// Mitsubishi GX Developer project: gate   PLC: FX1N

PROGRAM MAIN
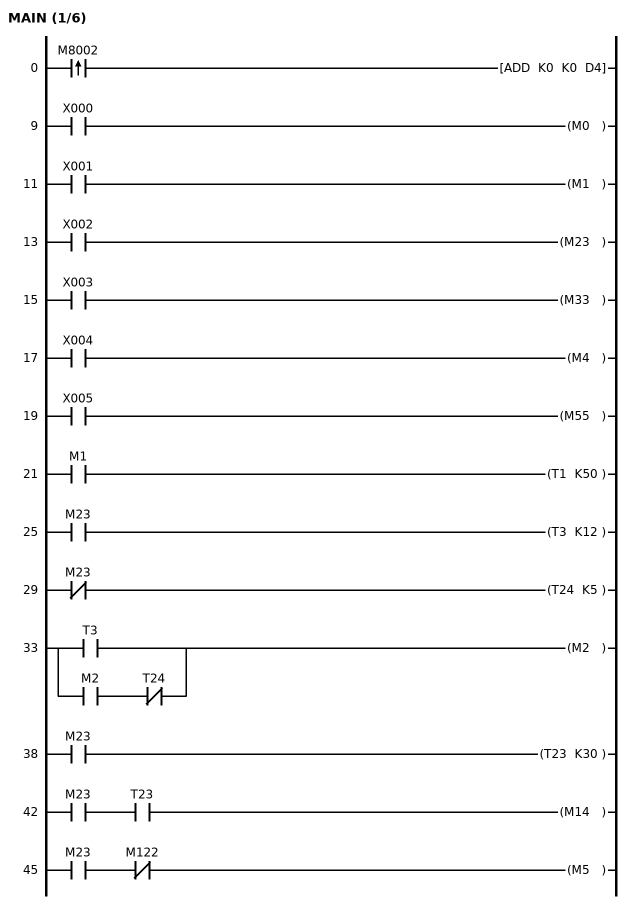
0     LDP     M8002
      ADD     K0 K0 D4
        [note] set car sensor to zero
9     LD      X000
      OUT     M0
        [note] external sw
11    LD      X001
      OUT     M1
        [note] internal sw
13    LD      X002
      OUT     M23
        [note] gate safety sw
15    LD      X003
      OUT     M33
        [note] car sensor
17    LD      X004
      OUT     M4
        [note] light on sensor
19    LD      X005
      OUT     M55
        [note] scrubber sensor
21    LD      M1
      OUT     T1 K50
        [note] internal open block delay
25    LD      M23
      OUT     T3 K12
        [note] X002 gate sensor
29    LDI     M23
      OUT     T24 K5
        [note] gate sensor debounse off
33    LD      T3
      LD      M2
      ANI     T24
      ORB
      OUT     M2
        [note] gate sensor debounce on
38    LD      M23
      OUT     T23 K30
        [note] car near gate timer
42    LD      M23
      AND     T23
      OUT     M14
        [note] car near gate
45    LD      M23
      ANI     M122
      OUT     M5
        [note] gate sensor and block
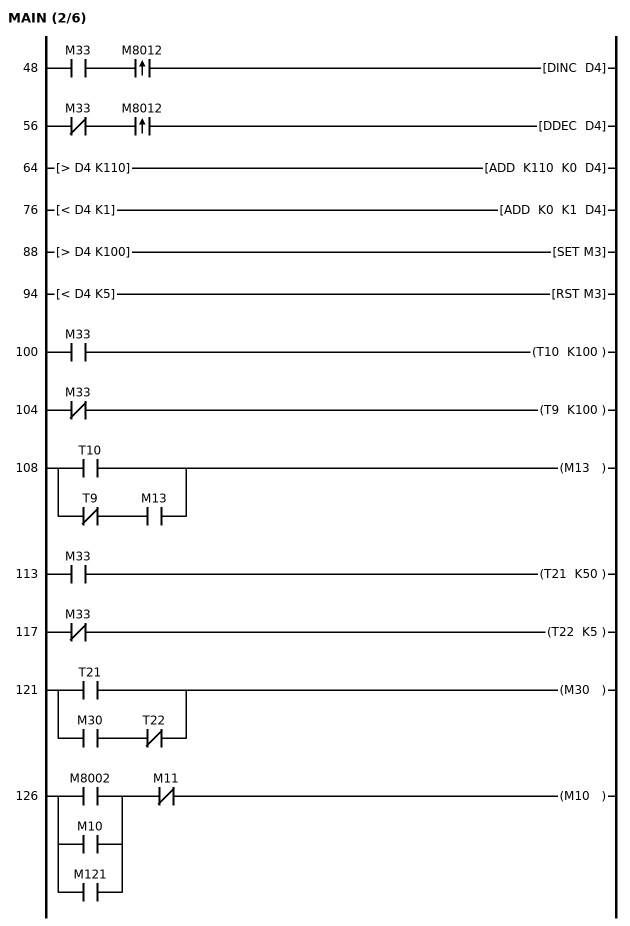
48    LD      M33
      ANDP    M8012
      DINC    D4
56    LDI     M33
      ANDP    M8012
      DDEC    D4
64    LD>     D4 K110
      ADD     K110 K0 D4
        [note] max limit  debounce car sensor
76    LD<     D4 K1
      ADD     K0 K1 D4
        [note] min limit  debounce car sensor
88    LD>     D4 K100
      SET     M3
94    LD<     D4 K5
      RST     M3
100   LD      M33
      OUT     T10 K100
        [note] x003  car sensor
104   LDI     M33
      OUT     T9 K100
        [note] debounce off
108   LD      T10
      LDI     T9
      AND     M13
      ORB
      OUT     M13
        [note] car sensor slow debounce
113   LD      M33
      OUT     T21 K50
        [note] car sensor fast  ON
117   LDI     M33
      OUT     T22 K5
        [note] car sensor fast OFF
121   LD      T21
      LD      M30
      ANI     T22
      ORB
      OUT     M30
        [note] car sensor fast
126   LD      M8002
      OR      M10
      OR      M121
      ANI     M11
      OUT     M10
        [note] ******** whaiting
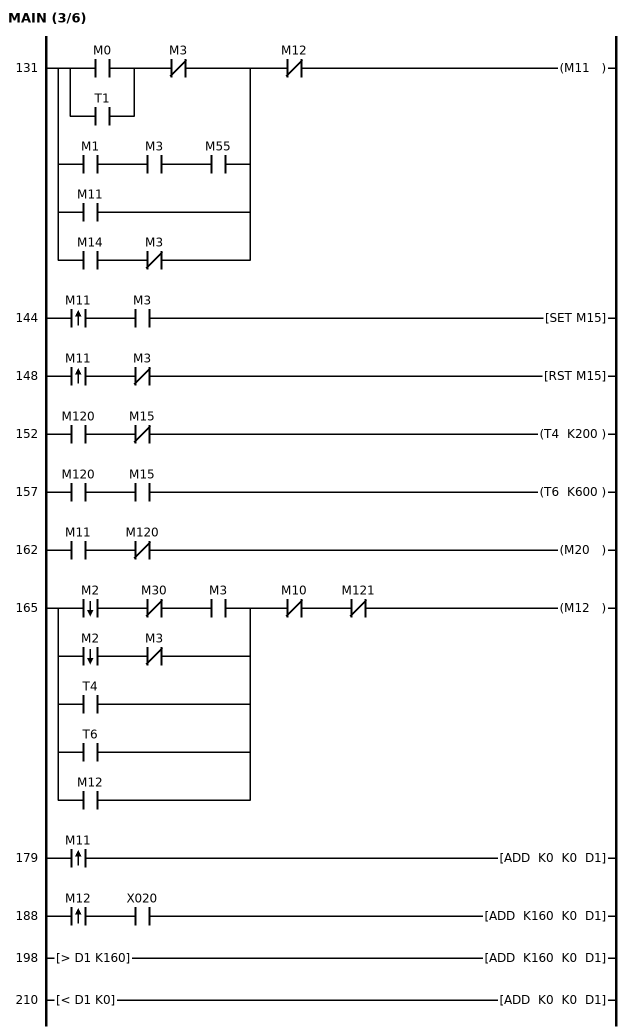
131   LD      M0
      OR      T1
      ANI     M3
      LD      M1
      AND     M3
      AND     M55
      ORB
      OR      M11
      LD      M14
      ANI     M3
      ORB
      ANI     M12
      OUT     M11
        [note] ******* entrance open begin
144   LDP     M11
      AND     M3
      SET     M15
        [note] car inside box
148   LDP     M11
      ANI     M3
      RST     M15
        [note] car outside box
152   LD      M120
      ANI     M15
      OUT     T4 K200
        [note] waiting entranñe
157   LD      M120
      AND     M15
      OUT     T6 K600
        [note] exit waiting
162   LD      M11
      ANI     M120
      OUT     M20
165   LDF     M2
      ANI     M30
      AND     M3
      LDF     M2
      ANI     M3
      ORB
      OR      T4
      OR      T6
      OR      M12
      ANI     M10
      ANI     M121
      OUT     M12
        [note] ******* entrance close begin
179   LDP     M11
      ADD     K0 K0 D1
        [note] set gate open start pos
188   LDP     M12
      AND     X020
      ADD     K160 K0 D1
        [note] set gate close start pos
198   LD>     D1 K160
      ADD     K160 K0 D1
        [note] gate up limit
210   LD<     D1 K0
      ADD     K0 K0 D1
        [note] gate close limit
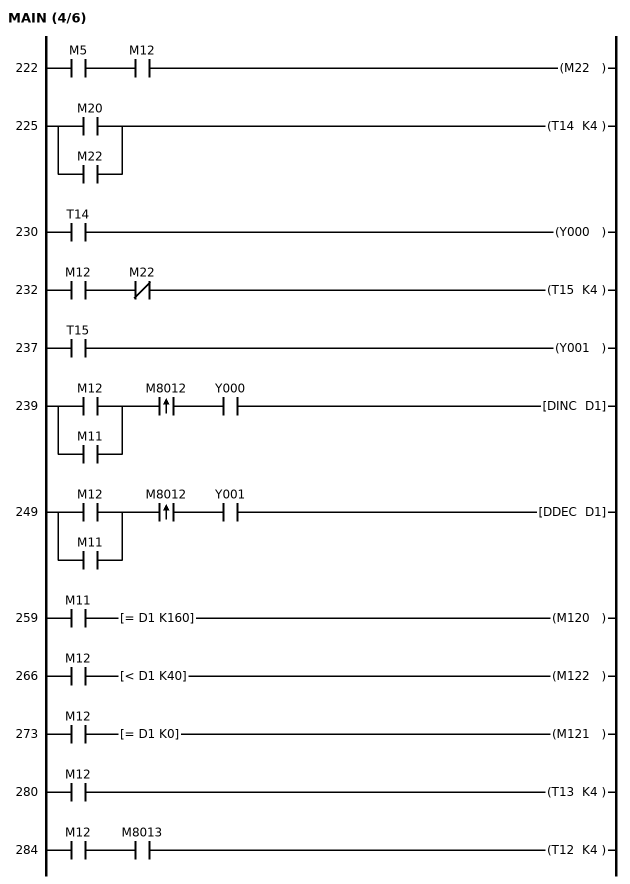
222   LD      M5
      AND     M12
      OUT     M22
        [note] open in close
225   LD      M20
      OR      M22
      OUT     T14 K4
        [note] gears safety time
230   LD      T14
      OUT     Y000
        [note] out relay block * open signal
232   LD      M12
      ANI     M22
      OUT     T15 K4
        [note] gears safety timer
237   LD      T15
      OUT     Y001
        [note] gate close output
239   LD      M12
      OR      M11
      ANDP    M8012
      AND     Y000
      DINC    D1
        [note] gate open timer incr
249   LD      M12
      OR      M11
      ANDP    M8012
      AND     Y001
      DDEC    D1
        [note] gate close timer decr
259   LD      M11
      AND=    D1 K160
      OUT     M120
        [note] open end
266   LD      M12
      AND<    D1 K40
      OUT     M122
        [note] block M5 and pic-pic
273   LD      M12
      AND=    D1 K0
      OUT     M121
        [note] close end
280   LD      M12
      OUT     T13 K4
        [note] close  pik
284   LD      M12
      AND     M8013
      OUT     T12 K4
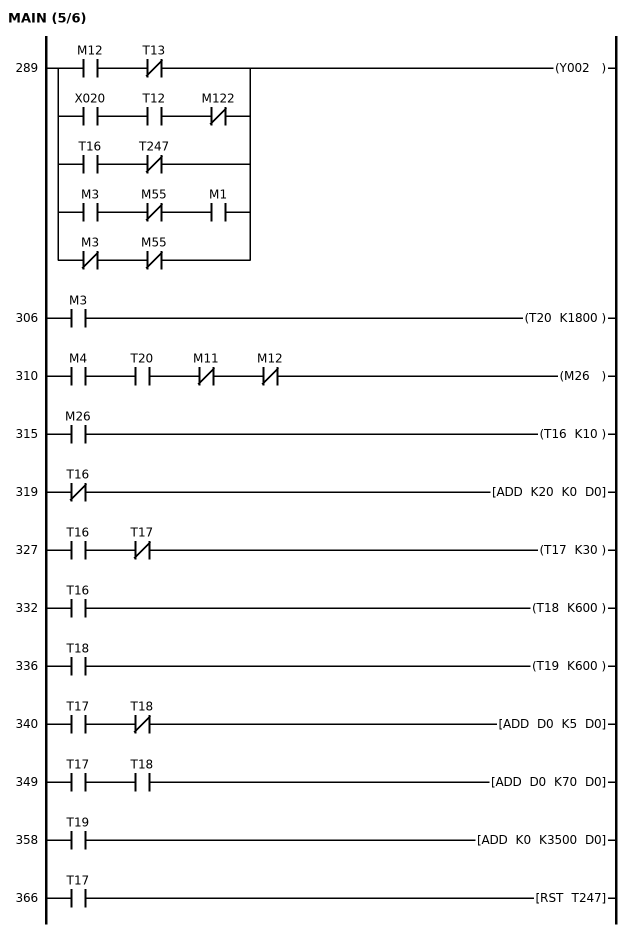
289   LD      M12
      ANI     T13
      LD      X020
      AND     T12
      ANI     M122
      ORB
      LD      T16
      ANI     T247
      ORB
      LD      M3
      ANI     M55
      AND     M1
      ORB
      LDI     M3
      ANI     M55
      ORB
      OUT     Y002
        [note] siren
306   LD      M3
      OUT     T20 K1800
        [note] block get-out entrance
310   LD      M4
      AND     T20
      ANI     M11
      ANI     M12
      OUT     M26
        [note] *** warning begin ****
315   LD      M26
      OUT     T16 K10
319   LDI     T16
      ADD     K20 K0 D0
327   LD      T16
      ANI     T17
      OUT     T17 K30
332   LD      T16
      OUT     T18 K600
        [note] 1 min timer
336   LD      T18
      OUT     T19 K600
340   LD      T17
      ANI     T18
      ADD     D0 K5 D0
349   LD      T17
      AND     T18
      ADD     D0 K70 D0
358   LD      T19
      ADD     K0 K3500 D0
366   LD      T17
      RST     T247
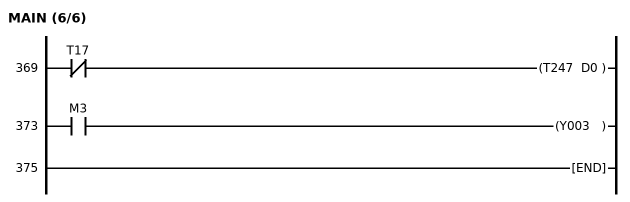
369   LDI     T17
      OUT     T247 D0
373   LD      M3
      OUT     Y003
        [note] svetofor
375   END
END_PROGRAM
